TYPE DUT_GroupStatus :
STRUCT
	Valid: BOOL;
	Busy: BOOL;
	GroupMoving: BOOL;
	GroupHoming: BOOL;
	GroupErrorStop: BOOL;
	GroupNotReady: BOOL;
	GroupStandby: BOOL;
	GroupStopping: BOOL;
	GroupDisabled: BOOL;
	AllAxesStanding: BOOL;
	InPosition: BOOL;
	Error: BOOL;
	ErrorID: UDINT;
END_STRUCT
END_TYPE

(* stored: Version 1.1.0.1
   DUT DUT_GroupStatus: Id {8da24330-28fc-457b-af4f-78411d1da7e7} *)
